FUNCTION_BLOCK MotorEnable
VAR_INPUT
END_VAR
VAR_OUTPUT
END_VAR
VAR
END_VAR

END_FUNCTION_BLOCK

(* stored: Version 1.1.0.1, ProductVersion 3.1.4024.11
   POU MotorEnable: Id {26c5168c-44be-4ae1-ba38-f4c46d49dcc5}, SpecialFunc None *)
